// TIA Portal V17 export
// export: Created 2025-03-10T13:11:51.3375822Z, ExportSetting WithDefaults, DisplayName Totally Integrated Automation Portal, DisplayVersion V17 Update 8, DisplayName TIA Portal Openness, DisplayVersion V17 Update 8, DisplayName TIA Portal Version Control Interface, DisplayVersion V17, DisplayName SINAMICS Startdrive Advanced, DisplayVersion V17 SP2, DisplayName SINAMICS Startdrive G110M, G120, G120C, G120D, G120P, G115D, DisplayVersion V17 SP2, DisplayName SINAMICS Startdrive G130, G150, S120, S150, SINAMICS MV, S210, DisplayVersion V17 SP2, DisplayName STEP 7 Professional, DisplayVersion V17 Update 8, DisplayName SINUMERIK ONE STEP 7 Toolbox, DisplayVersion V17 Update 12, DisplayName SINUMERIK 840D sl STEP 7 Toolbox, DisplayVersion V17 Update 12, DisplayName STEP 7 Safety, DisplayVersion V17 Update 6, DisplayName WinCC Advanced, DisplayVersion V17 Update 8
VAR_GLOBAL   // PLC tag table "TAGS_IO_GENERAL_CLADDING"
   "/////_MODES_/////" AT %M6050.0 : Bool;   // /////_MODES_/////
   BA_MODES_BA1_BUTTON_I AT %M6050.1 : Bool;   // BA MODES BA1 MODE BUTTON INPUT
   BA_MODES_BA2_BUTTON_I AT %M6050.2 : Bool;   // BA MODES BA2 MODE BUTTON INPUT
   BA_MODES_BA3_BUTTON_I AT %M6050.3 : Bool;   // BA MODES BA3 MODE BUTTON INPUT
   BA_MODES_BA1_LED_Q AT %M6050.4 : Bool;   // BA MODES BA1 MODE BUTTON LED OUTPUT
   BA_MODES_BA2_LED_Q AT %M6050.5 : Bool;   // BA MODES BA2 MODE BUTTON LED OUTPUT
   BA_MODES_BA3_LED_Q AT %M6050.6 : Bool;   // BA MODES BA3 MODE BUTTON LED OUTPUT
   "/////_CRM_/////" AT %M6060.0 : Bool;   // /////_CRM_/////
   CONTROL_ON_I AT %I37.1 : Bool;   // CONTROL ON INPUT
   MACHINE_ON_STP_SRV_DEL_Q AT %M6060.3 : Bool;   // MACHINE ON STOP SERVICES DELAYED OUTPUT
   "/////_POWER_SUPPLY_/////" AT %M6080.0 : Bool;   // /////_POWER_SUPPLY_/////
   INFEED_MODULE_1_READY_I AT %I35.0 : Bool;   // INFEED MODULE 1 READY INPUT
   INFEED_MODULE_1_ON_I AT %I35.1 : Bool;   // INFEED MODULE 1 ON INPUT
   INFEED_MODULE_1_OVRTM_I AT %M6080.3 : Bool;   // INFEED MODULE 1 OVERTEMPERATURE INPUT
   INFEED_MODULE_OFF3_Q AT %Q32.1 : Bool;   // INFEED MODULE OFF 3 OUTPUT
   INFEED_MODULE_ON_OFF_Q AT %Q32.0 : Bool;   // INFEED MODULE ON OFF OUTPUT
   INFEED_MODULE_2_READY_I AT %M6080.6 : Bool;   // INFEED MODULE 2 READY INPUT
   INFEED_MODULE_2_ON_I AT %M6080.7 : Bool;   // INFEED MODULE 2 ON INPUT
   INFEED_MODULE_2_OVRTM_I AT %M6081.0 : Bool;   // INFEED MODULE 2 OVERTEMPERATURE INPUT
   INFEED_MODULE_2_OFF3_Q AT %M6081.1 : Bool;   // INFEED MODULE 2 OFF 3 OUTPUT
   INFEED_MODULE_2_ON_OFF_Q AT %M6081.2 : Bool;   // INFEED MODULE 2 ON OFF OUTPUT
   "/////_ELECTRICAL_CABINET_/////" AT %M6100.0 : Bool;   // /////_ELECTRICAL_CABINET_/////
   MAIN_CIRCUIT_BREAKER_I AT %I32.2 : Bool;   // MAIN CABINET CIRCUIT BREAKER TRIPPED INPUT
   MAIN_SWITCH_INPUT AT %M6100.2 : Bool;   // ELECTRICAL CABINET MAIN SWITCH INPUT
   ETHERNET_SWITCH_1_FAULT_I AT %I38.0 : Bool;   // ETHERNET SWITCH 1 FAULT INPUT
   ETHERNET_SWITCH_2_FAULT_I AT %I38.1 : Bool;   // ETHERNET SWITCH 2 FAULT INPUT
   ETHERNET_SWITCH_3_FAULT_I AT %I38.2 : Bool;   // ETHERNET SWITCH 3 FAULT INPUT
   ETHERNET_SWITCH_4_FAULT_I AT %I38.4 : Bool;   // ETHERNET SWITCH 4 FAULT INPUT
   AIR_UNIT_1_OK_SEOC AT %M6101.0 : Bool;   // AIR UNIT 1 OK INPUT
   AIR_UNIT_2_OK_SEOC AT %M6101.1 : Bool;   // AIR UNIT 2 OK INPUT
   AIR_UNIT_1_BREAKER_SEOC AT %M6101.2 : Bool;   // AIR UNIT 1 BREAKER INPUT
   AIR_UNIT_2_BREAKER_SEOC AT %M6101.3 : Bool;   // AIR UNIT 2 BREAKER INPUT
   CIRCUIT_BREAKER_1_24_VDC AT %I33.4 : Bool;   // CIRCUIT BREAKER 1 24 V DC INPUT
   CIRCUIT_BREAKER_2_24_VDC AT %I33.5 : Bool;   // CIRCUIT BREAKER 2 24 V DC INPUT
   I_OVER_VOLTAGE AT %M6101.6 : Bool;   // OVER VOLTAGE INPUT
   I_BREAKER_QFC03 AT %I32.6 : Bool;   // BREAKER FC03 INPUT
   PS_24V_NOT_READY_DEV_1_I AT %I34.0 : Bool;   // POWER SUPPLY 24V NOT READY DEVICE 1 INPUT
   PS_24V_NOT_READY_DEV_2_I AT %I34.1 : Bool;   // POWER SUPPLY 24V NOT READY DEVICE 2 INPUT
   PS_24V_NOT_READY_DEV_3_I AT %I34.2 : Bool;   // POWER SUPPLY 24V NOT READY DEVICE 3 INPUT
   PS_24V_NOT_READY_DEV_4_I AT %I34.3 : Bool;   // POWER SUPPLY 24V NOT READY DEVICE 4 INPUT
   PS_24V_NOT_READY_DEV_5_I AT %I34.4 : Bool;   // POWER SUPPLY 24V NOT READY DEVICE 5 INPUT
   PS_24V_NOT_READY_DEV_6_I AT %I34.5 : Bool;   // POWER SUPPLY 24V NOT READY DEVICE 6 INPUT
   FAULT_PS_I AT %M6102.4 : Bool;   // FAULT POWER SUPPLY INPUT
   SINAMICS_CIRC_BREAKER_I AT %I33.2 : Bool;   // SINAMICS CIRCUIT BREAKER TRIPPED INPUT
   BATTERY_OK_I AT %M6102.6 : Bool;   // INPUT BATTERY OK SITOP UPS500S
   PS_24V_BKR_DEV_1_I AT %M6103.0 : Bool;   // POWER SUPPLY 24V CIRCUIT BREAKER TRIPPED DEVICE 1 INPUT (WITHOUT FB)
   PS_24V_BKR_DEV_2_I AT %M6103.1 : Bool;   // POWER SUPPLY 24V CIRCUIT BREAKER TRIPPED DEVICE 2 INPUT (WITHOUT FB)
   PS_24V_BKR_DEV_3_I AT %M6103.2 : Bool;   // POWER SUPPLY 24V CIRCUIT BREAKER TRIPPED DEVICE 3 INPUT (WITHOUT FB)
   PS_24V_BKR_DEV_4_I AT %M6103.3 : Bool;   // POWER SUPPLY 24V CIRCUIT BREAKER TRIPPED DEVICE 4 INPUT (WITHOUT FB)
   DIAGNOSIS_MOD1_I AT %M6103.4 : Bool;   // DIAGNOSIS MODULE 1 INPUT(WITH FB)
   DIAGNOSIS_MOD2_I AT %M6103.5 : Bool;   // DIAGNOSIS MODULE 2 INPUT(WITH FB)
   DIAGNOSIS_MOD3_I AT %M6103.6 : Bool;   // DIAGNOSIS MODULE 3 INPUT(WITH FB)
   DIAGNOSIS_MOD4_I AT %M6103.7 : Bool;   // DIAGNOSIS MODULE 4 INPUT(WITH FB)
   CIRCUIT_BREAKER_120VAC_I AT %M6104.0 : Bool;   // CIRCUIT BREAKER F1 - F4 INPUT
   CB_CABINET_LIGHTING_I AT %M6104.1 : Bool;   // CIRCUIT BREAKER CABINET LIGHTING INPUT
   I_BREAKER_WAT AT %M6104.2 : Bool;   // INPUT BREAKER SENTRON PAC3200
   CB_JIB_CRANE_I AT %M6104.3 : Bool;   // CIRCUIT BREAKER JIB CRANE INPUT
   ELEC_CAB_DOOR_CLOSED_I AT %I37.4 : Bool;   // INPUT ELECTRICAL CABINET DOOR CLOSED
   "/////_MPP_AND_SIGNAL_TOWER_/////" AT %M6120.0 : Bool;   // /////_MPP_AND_SIGNAL_TOWER_/////
   SIGNAL_TWR_RED_LIGHT_Q AT %Q39.2 : Bool;   // SIGNAL TOWER RED LIGHT OUTPUT
   SIGNAL_TWR_GREEN_LIGHT_Q AT %Q39.0 : Bool;   // SIGNAL TOWER GREEN LIGHT OUTPUT
   SIGNAL_TWR_ORANGE_LIGHT_Q AT %Q39.1 : Bool;   // SIGNAL TOWER ORANGE LIGHT OUTPUT
   SIGNAL_TWR_HOOTER_Q AT %M6120.5 : Bool;   // SIGNAL TOWER HOOTER LIGHT OUTPUT
   MPP_BYPASS_GATES_I AT %I41.1 : Bool;   // MAIN PANEL BYPASS GATES INPUT
   MACH_LIGHT_SELECTOR_ON_I AT %I41.0 : Bool;   // MACHINE LIGHT SELECTOR ON INPUT
   AUX_OP_PANEL_START_CYCLE_LAMP AT %Q40.7 : Bool;   // AUX OP PANEL START CYCLE LAMP
   MACH_LIGHT_ON_1_Q AT %Q32.6 : Bool;   // MACHINE LIGHT ON 1 OUTPUT
   MACH_LIGHT_ON_2_Q AT %M6128.3 : Bool;   // MACHINE LIGHT ON 2 OUTPUT
   MACHINE_ON_Q AT %Q32.4 : Bool;   // MACHINE ON OUTPUT
   MASCHINE_AUS_Q AT %Q32.2 : Bool;   // MACHINE OFF AUX PANEL OUTPUT
   MASCHINE_EIN_Q AT %Q32.3 : Bool;   // MACHINE ON AUX PANEL OUTPUT
   "/////_SAFETY_DOORS_/////" AT %M6180.0 : Bool;   // /////_SAFETY_DOORS_/////
   UNIT_01_ST02_SAFE_DR_CLSD_I AT %I60.2 : Bool;   // UNIT 01 ST02 SAFETY DOOR CLOSED INPUT
   UNIT_01_ST02_SAFE_DR_UNLOCK_Q AT %Q60.2 : Bool;   // UNIT 01 ST02 SAFETY DOOR UNLOCK OUTPUT
   UNIT_01_ST02_SAFE_DR_RED_L_Q AT %M6180.3 : Bool;   // UNIT 01 ST02 SAFETY DOOR RED LIGTH OUTPUT
   UNIT_01_ST02_SAFE_DR_GREEN_L_Q AT %M6180.4 : Bool;   // UNIT 01 ST02 SAFETY DOOR GREEN LIGTH OUTPUT
   UNIT_01_MAIN_SAFE_DR_CLSD_I AT %I60.0 : Bool;   // UNIT 01 MAIN SAFETY DOOR CLOSED INPUT
   UNIT_01_MAIN_SAFE_DR_UNLOCK_Q AT %Q60.0 : Bool;   // UNIT 01 MAIN SAFETY DOOR UNLOCK OUTPUT
   UNIT_01_MAIN_SAFE_DR_RED_L_Q AT %M6181.3 : Bool;   // UNIT 01 MAIN SAFETY DOOR RED LIGTH OUTPUT
   UNIT_01_MAIN_SAFE_DR_GREEN_L_Q AT %M6181.4 : Bool;   // UNIT 01 MAIN SAFETY DOOR GREEN LIGTH OUTPUT
   UNIT_01_ST04_SAFE_DR_CLSD_I AT %I60.1 : Bool;   // UNIT 01 ST04 SAFETY DOOR CLOSED INPUT
   UNIT_01_ST04_SAFE_DR_UNLOCK_Q AT %Q60.1 : Bool;   // UNIT 01 ST04 SAFETY DOOR UNLOCK OUTPUT
   UNIT_01_ST04_SAFE_DR_RED_L_Q AT %M6180.7 : Bool;   // UNIT 01 ST04 SAFETY DOOR RED LIGTH OUTPUT
   UNIT_01_ST04_SAFE_DR_GREEN_L_Q AT %M6181.0 : Bool;   // UNIT 01 ST04 SAFETY DOOR GREEN LIGTH OUTPUT
   UNIT_01_MAINT_SAFE_DR_CLSD_I AT %M6181.5 : Bool;   // UNIT 01 MAINTENANCE SAFETY DOOR CLOSED INPUT
   UNIT_01_MAINT_SAFE_DR_UNLOCK_Q AT %M6181.6 : Bool;   // UNIT 01 MAINTENANCE SAFETY DOOR UNLOCK OUTPUT
   UNIT_01_MAINT_SAFE_DR_RED_L_Q AT %M6181.7 : Bool;   // UNIT 01 MAINTENANCE SAFETY DOOR RED LIGTH OUTPUT
   UNIT_01_MAINT_SAFE_DR_GREEN_L_Q AT %M6182.0 : Bool;   // UNIT 01 MAINTENANCE SAFETY DOOR GREEN LIGTH OUTPUT
   UNIT_01_OERLIKON_SAFE_DR_CLSD_I AT %M6182.1 : Bool;   // UNIT 01 OERLIKON SAFETY DOOR CLOSED INPUT
   UNIT_01_OERLIKON_SAFE_DR_UNLOCK_Q AT %M6182.2 : Bool;   // UNIT 01 OERLIKON SAFETY DOOR UNLOCK OUTPUT
   UNIT_01_OERLIKON_SAFE_DR_RED_L_Q AT %M6182.5 : Bool;   // UNIT 01 OERLIKON SAFETY DOOR RED LIGTH OUTPUT
   UNIT_01_OERLIKON_SAFE_DR_GREEN_L_Q AT %M6182.6 : Bool;   // UNIT 01 OERLIKON SAFETY DOOR GREEN LIGTH OUTPUT
   UNIT_02_ST02_SAFE_DR_CLSD_I AT %I1060.0 : Bool;   // UNIT 02 ST02 SAFETY DOOR CLOSED INPUT
   UNIT_02_ST02_SAFE_DR_UNLOCK_Q AT %Q1060.0 : Bool;   // UNIT 02 ST02 SAFETY DOOR UNLOCK OUTPUT
   UNIT_02_ST02_SAFE_DR_RED_L_Q AT %M6182.3 : Bool;   // UNIT 02 ST02 SAFETY DOOR RED LIGTH OUTPUT
   UNIT_02_ST02_SAFE_DR_GREEN_L_Q AT %M6182.4 : Bool;   // UNIT 02 ST02 SAFETY DOOR GREEN LIGTH OUTPUT
   UNIT_02_MAIN_SAFE_DR_CLSD_I AT %I1060.1 : Bool;   // UNIT 02 MAIN SAFETY DOOR CLOSED INPUT
   UNIT_02_MAIN_SAFE_DR_UNLOCK_Q AT %Q1060.1 : Bool;   // UNIT 02 MAIN SAFETY DOOR UNLOCK OUTPUT
   UNIT_02_MAIN_SAFE_DR_RED_L_Q AT %M6182.7 : Bool;   // UNIT 02 FRONT SAFETY DOOR RED LIGTH OUTPUT
   UNIT_02_MAIN_SAFE_DR_GREEN_L_Q AT %M6183.0 : Bool;   // UNIT 02 FRONT SAFETY DOOR GREEN LIGTH OUTPUT
   UNIT_02_ST04_SAFE_DR_CLSD_I AT %I1060.2 : Bool;   // UNIT 02 ST04 SAFETY DOOR CLOSED INPUT
   UNIT_02_ST04_SAFE_DR_UNLOCK_Q AT %Q1060.2 : Bool;   // UNIT 02 ST04 SAFETY DOOR UNLOCK OUTPUT
   UNIT_02_ST04_SAFE_DR_RED_L_Q AT %M6183.3 : Bool;   // UNIT 02 ST04 SAFETY DOOR RED LIGTH OUTPUT
   UNIT_02_ST04_SAFE_DR_GREEN_L_Q AT %M6183.4 : Bool;   // UNIT 02 ST04 SAFETY DOOR GREEN LIGTH OUTPUT
   UNIT_02_MAINT_SAFE_DR_CLSD_I AT %M6183.5 : Bool;   // UNIT 02 MAINTENANCE SAFETY DOOR CLOSED INPUT
   UNIT_02_MAINT_SAFE_DR_UNLOCK_Q AT %M6183.6 : Bool;   // UNIT 02 MAINTENANCE SAFETY DOOR UNLOCK OUTPUT
   UNIT_02_MAINT_SAFE_DR_RED_L_Q AT %M6183.7 : Bool;   // UNIT 02 MAINTENANCE SAFETY DOOR RED LIGTH OUTPUT
   UNIT_02_MAINT_SAFE_DR_GREEN_L_Q AT %M6184.0 : Bool;   // UNIT 02 MAINTENANCE SAFETY DOOR GREEN LIGTH OUTPUT
   UNIT_02_OERLIKON_SAFE_DR_CLSD_I AT %M6183.1 : Bool;   // UNIT 02 OERLIKON SAFETY DOOR CLOSED INPUT
   UNIT_02_OERLIKON_SAFE_DR_UNLOCK_Q AT %M6183.2 : Bool;   // UNIT 02 OERLIKON SAFETY DOOR UNLOCK OUTPUT
   UNIT_02_OERLIKON_SAFE_DR_RED_L_Q AT %M6184.1 : Bool;   // UNIT 02 OERLIKON SAFETY DOOR RED LIGTH OUTPUT
   UNIT_02_OERLIKON_SAFE_DR_GREEN_L_Q AT %M6184.2 : Bool;   // UNIT 02 OERLIKON SAFETY DOOR GREEN LIGTH OUTPUT
   "/////_OTHER_CIRCUIT_BREAKERS_/////" AT %M8308.0 : Bool;   // /////_OTHER_CIRCUIT_BREAKERS_/////
   LASER_U01_CIRCUIT_BREAKER_TRIPPED AT %I32.4 : Bool;   // LASER SOURCE UNIT 01 CIRCUIT BREEAKER TRIPPED
   LASER_U02_CIRCUIT_BREAKER_TRIPPED AT %I32.5 : Bool;   // LASER SOURCE UNIT 02 CIRCUIT BREEAKER TRIPPED
   ROBOT_CELL_CIRCUIT_BREAKER_TRIPPED AT %I33.0 : Bool;   // ROBOT CELL CIRCUIT BREAKER TRIPPED
   QB23_CIRCUIT_BREAKER_24_VDC_INPUT AT %I33.1 : Bool;   // QB23 CIRCUIT BREEAKER 24 VDC INPUT
   HEATER_CIRCUIT_BREAKER_TRIPPED AT %M8308.5 : Bool;   // HEATER CIRCUIT BREAKER TRIPPED
   PC_CABINET_CIRCUIT_BREAKER_TRIPPED AT %I35.2 : Bool;   // CHILLER CIRCUIT BREAKER TRIPPED
   OERLIKON_U01_CIRCUIT_BREAKER_TRIPPED AT %M8308.3 : Bool;   // OERLIKON UNIT 01 CIRCUIT BREEAKER TRIPPED
   OERLIKON_U02_CIRCUIT_BREAKER_TRIPPED AT %M8308.4 : Bool;   // OERLIKON UNIT 02 CIRCUIT BREEAKER TRIPPED
   STIRRER_CIRCUIT_BREAKER_TRIPPED AT %M8309.1 : Bool;   // STIRRRER CIRCUIT BREAKER TRIPPED
   CHILLER_CIRCUIT_BREAKER_TRIPPED AT %M8309.2 : Bool;   // CHILLER CIRCUIT BREAKER TRIPPED
   HOPPER_CIRCUIT_BREAKER_TRIPPED AT %M8309.3 : Bool;   // HOPPER CIRCUIT BREAKER TRIPPERD
   COOLING_UNIT_CIRCUIT_BREAKER AT %I32.3 : Bool;   // COOLING UNIT CIRCUIT BREAKER
   SINAMICS_CIRCUIT_BREAKER_TRIPPED AT %M6101.7 : Bool;   // SINAMICS CIRCUIT BREAKER TRIPPED
   WATTMETER_BREAKER_I AT %I32.0 : Bool;   // WATTMETER BREAKER INPUT
   I_BREAKER_QB02 AT %I32.7 : Bool;   // BREAKER QB02 INPUT
   "0FC20_CIRCUIT_BREAKER_TRIPPED_I" AT %I39.0 : Bool;   // 0FC20 CIRCUIT BREAKER TRIPPED INPUT
   "0FC22_CIRCUIT_BREAKER_TRIPPED_I" AT %I39.2 : Bool;   // 0FC22 CIRCUIT BREAKER TRIPPED INPUT
   "0FC23_CIRCUIT_BREAKER_TRIPPED_I" AT %I39.3 : Bool;   // 0FC23 CIRCUIT BREAKER TRIPPED INPUT
   "0FC21_CIRCUIT_BREAKER_TRIPPED_I" AT %I39.1 : Bool;   // 0FC21 CIRCUIT BREAKER TRIPPED INPUT
   "/////_LINE_CONTACTOR_/////" AT %M6200.0 : Bool;   // /////_LINE_CONTACTOR_/////
   LINE_CONTACTOR_FDBCK_1_I AT %M6200.1 : Bool;   // LINE CONTACTOR FEEDBACK 1 INPUT
   LINE_CONTACTOR_FDBCK_2_I AT %M6200.2 : Bool;   // LINE CONTACTOR FEEDBACK 2 INPUT
   LINE_CONTACTOR_ON_1_Q AT %M6200.3 : Bool;   // LINE CONTACTOR ON 1 OUTPUT
   LINE_CONTACTOR_ON_2_Q AT %M6200.4 : Bool;   // LINE CONTACTOR ON 2 OUTPUT
   CONTROL_VOLTAGE_ON_I AT %I37.0 : Bool;   // CONTROL VOLTAGE ON
   ELECTRICAL_CABINET_OVERTEMP_I AT %I37.7 : Bool;   // ELECTRICAL CABINET OVERTEMPERATURE INPUT NO
   BATTERY_ALARM_I AT %M6102.7 : Bool;   // INPUT BATTERY ALARM SITOP UPS500S
   PILZ_ESTOP_OK_I AT %M6102.1 : Bool;   // PILZ EMERGENCY STOP OK INPUT NO
   BATTERY_85_I AT %M6104.5 : Bool;   // INPUT BATTERY 85% SITOP UPS500S
   "/////_OTHER_CONTACTOR_/////" AT %M8309.5 : Bool;   // /////_OTHER_CONTACTOR_/////
   DRIVES_MAIN_CONTACTOR AT %Q33.0 : Bool;   // DRIVES SWITCH ON MAIN CONTACTOR
   LASER_SOURCE_ENABLE_1 AT %Q42.4 : Bool;   // LASER SOURCE ENABLE 1
   LASER_SOURCE_ENABLE_2 AT %Q42.5 : Bool;   // LASER SOURCE ENABLE 2
   PN_DELETE_DATA_Q AT %Q33.5 : Bool;   // PN-DELETE DATA OUTPUT
   PN_ANALYSE_START_STOP_Q AT %Q33.6 : Bool;   // PN-ANALYSE START/STOP OUTPUT
   PN_ANALYSE_ACKNOWLEDGE_Q AT %Q33.7 : Bool;   // PN-ANALYSE ACKNOWLEDGE OUTPUT
   LASER_UNIT_01_OK AT %I45.2 : Bool;   // LASER UNIT 01 OK
   LASER_UNIT_02_OK AT %I45.3 : Bool;   // LASER UNIT 02 OK
   "/////_POWER_ON_BALLUFF_SUBMODULES_/////" AT %M8312.0 : Bool;
   KF470_BALLUFF_SUBMODULE_ON AT %Q81.3 : Bool;   // KF470 BALLUFF SUBMODULE ON
   KF480_BALLUFF_SUBMODULE_ON AT %Q81.4 : Bool;   // KF480 BALLUFF SUBMODULE ON
   KF490_BALLUFF_SUBMODULE_ON AT %Q81.5 : Bool;   // KF490 BALLUFF SUBMODULE ON
   KF500_BALLUFF_SUBMODULE_ON AT %Q81.6 : Bool;   // KF500 BALLUFF SUBMODULE ON
   KF570_BALLUFF_SUBMODULE_ON AT %Q71.5 : Bool;   // KF570 BALLUFF SUBMODULE ON
   KF578_BALLUFF_SUBMODULE_ON AT %Q71.6 : Bool;   // KF578 BALLUFF SUBMODULE ON
   KF1470_BALLUFF_SUBMODULE_ON AT %Q1081.3 : Bool;   // KF1470 BALLUFF SUBMODULE ON
   KF1480_BALLUFF_SUBMODULE_ON AT %Q1081.4 : Bool;   // KF1480 BALLUFF SUBMODULE ON
   KF1490_BALLUFF_SUBMODULE_ON AT %Q1081.5 : Bool;   // KF1490 BALLUFF SUBMODULE ON
   KF1500_BALLUFF_SUBMODULE_ON AT %Q1081.6 : Bool;   // KF1500 BALLUFF SUBMODULE ON
   KF1570_BALLUFF_SUBMODULE_ON AT %Q1074.5 : Bool;   // KF1570 BALLUFF SUBMODULE ON
   KF1578_BALLUFF_SUBMODULE_ON AT %Q1074.6 : Bool;   // KF1578 BALLUFF SUBMODULE ON
   MACHINE_OFF_I AT %I41.3 : Bool;   // MACHINE OFF AUX PANEL INPUT
   U01_TURN_CONTROL_2 AT %I500.5 : Bool;   // UNIT 01 TURN CONTROL 2
   U01_TURN_CONTROL_1 AT %I500.4 : Bool;   // UNIT 01 TURN CONTROL 1
   CIRCUIT_BREAKER_TRIPPED_LIGHT_STA_3 AT %I39.4 : Bool;   // CIRCUIT BREAKER TRIPPED LIGHT STATION 3 INPUT
   PROFINET_CONTROL_UNIT_FAULT_I AT %I38.3 : Bool;   // PROFINET CONTROL UNIT FAULT INPUT
   I_CAMERAS_BREAKER_0FC30 AT %I33.6 : Bool;   // CAMERAS BREAKER 0FC30 INPUT
   COOLING_SYSTEM_BUFFER_CIRCUIT_BREAKER_TRIPPED AT %I37.3 : Bool;   // COOLING SYSTEM FOR COOLING BUFFER CIRCUIT BREAKER TRIPPED
   COOLING_SYSTEM_MACHINE_CIRCUIT_BREAKER_TRIPPED AT %I37.2 : Bool;   // COOLING SYSTEM FOR MACHINE CIRCUIT BREAKER TRIPPED
END_VAR
